(* Logix 5000 project; controller cal1632 1756-L62 rev 16.20; software revision 16.05; part 46 of 57 *)
(* tags used below, declared in another part *)
   FAULT : BOOL;
   HMI : BOOL;
   p01_recipe_active : recipe;
   p01r09_pb_global_reset : BOOL;
   p26_ao_dia_a : REAL;
   p26_ao_dia_b : REAL;
   p26_inactive_tension_sp : REAL;
   p26r03_upper_A_tension_on : BOOL;
   p26r03_upper_B_tension_on : BOOL;
   p26r10 : routine;
   p26r10_timer_fault : TIMER[4];
   p26r10_timer_warning : TIMER[4];
   p26r10_ula_selected_tension : REAL;
   p26r10_ulb_selected_tension : REAL;
   p26r10_unwind_a_brake_torque : REAL;
   p26r10_unwind_a_dia_ft : REAL;
   p26r10_unwind_b_brake_torque : REAL;
   p26r10_unwind_b_dia_ft : REAL;
   p27_ao_dia_a : REAL;
   p27_ao_dia_b : REAL;
   p27_dint_to_hmi : DINT[16];
   p27_lft_a_prs_input_max : REAL;
   p27_lft_a_prs_input_min : REAL;
   p27_lft_a_prs_output_max : REAL;
   p27_lft_a_prs_output_min : REAL;
   p27_lft_b_prs_input_max : REAL;
   p27_lft_b_prs_input_min : REAL;
   p27_lft_b_prs_output_max : REAL;
   p27_lft_b_prs_output_min : REAL;
   p27_lla_prs_input_max : REAL;
   p27_lla_prs_input_min : REAL;
   p27_lla_prs_output_max : REAL;
   p27_lla_prs_output_min : REAL;
   p27_lla_prs_scp : SYS_SCP;
   p27_llb_prs_input_max : REAL;
   p27_llb_prs_input_min : REAL;
   p27_llb_prs_output_max : REAL;
   p27_llb_prs_output_min : REAL;
   p27_llb_prs_scp : SYS_SCP;
   p27r01 : routine;
   p27r02 : routine;
   p27r02_fault_exists : BOOL;
   p27r02_timer_fault : TIMER[4];
   p27r02_timer_warning : TIMER[4];
   p27r02_unack_fault : BOOL;
   p27r02_unack_warning : BOOL;
   p27r02_warning_exists : BOOL;
   p27r03 : routine;
   p27r03_a_radius : REAL;
   p27r03_ai_dia_a_sensor : REAL;
   p27r03_ai_dia_b_sensor : REAL;
   p27r03_b_radius : REAL;
   p27r03_lower_A_tension_on : BOOL;
   p27r03_lower_B_tension_on : BOOL;
   p27r03_ltf_a_diameter_scp : SYS_SCP;
   p27r03_ltf_b_diameter_scp : SYS_SCP;
   p27r03_timer_fault : TIMER[4];
   p27r03_timer_warning : TIMER[4];
   p27r03_winder_a_distance : REAL;
   p27r03_winder_b_distance : REAL;
   p27r04 : routine;
   p27r04_timer_fault : TIMER[4];
   p27r04_timer_warning : TIMER[4];
   p27r05 : routine;
   p27r05_timer_fault : TIMER[4];
   p27r05_timer_warning : TIMER[4];
   p27r06 : routine;
   p27r07 : routine;
   p27r08 : routine;
   p27r09 : routine;
   p27r10 : routine;
   p27r10_lla_selected_tension : REAL;
   p27r10_llb_selected_tension : REAL;
   p27r11 : routine;
(* P26_Upper_Poly_Letoff, continued *)

ROUTINE R10_Tension_A   (* ladder *)
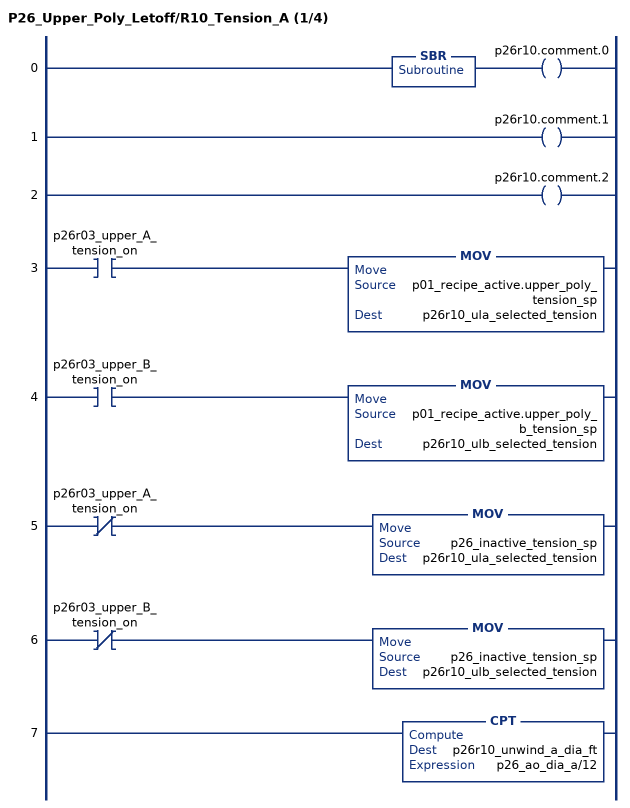
   0: SBR()OTE(p26r10.comment.0);
   1: OTE(p26r10.comment.1);
   2: OTE(p26r10.comment.2);
   3: XIC(p26r03_upper_A_tension_on)MOV(p01_recipe_active.upper_poly_tension_sp,p26r10_ula_selected_tension);
   4: XIC(p26r03_upper_B_tension_on)MOV(p01_recipe_active.upper_poly_b_tension_sp,p26r10_ulb_selected_tension);
   5: XIO(p26r03_upper_A_tension_on)MOV(p26_inactive_tension_sp,p26r10_ula_selected_tension);
   6: XIO(p26r03_upper_B_tension_on)MOV(p26_inactive_tension_sp,p26r10_ulb_selected_tension);
   7: CPT(p26r10_unwind_a_dia_ft,p26_ao_dia_a/12);
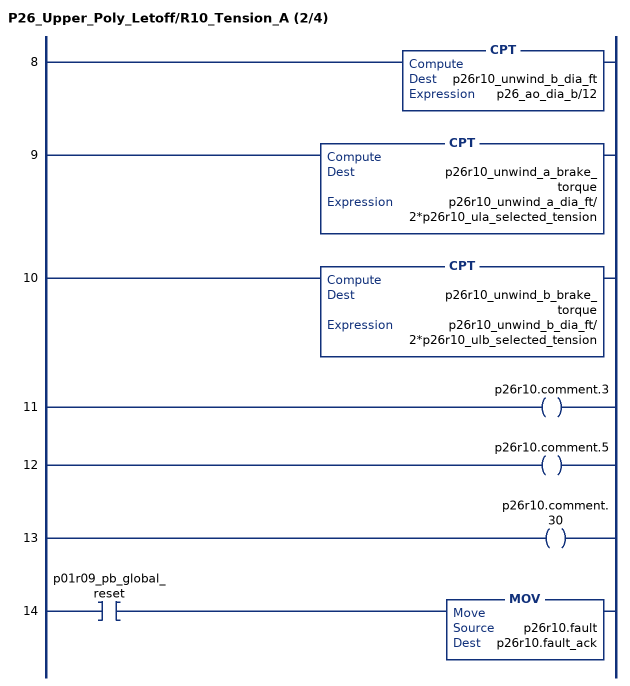
   8: CPT(p26r10_unwind_b_dia_ft,p26_ao_dia_b/12);
   9: CPT(p26r10_unwind_a_brake_torque,p26r10_unwind_a_dia_ft/2*p26r10_ula_selected_tension);
   10: CPT(p26r10_unwind_b_brake_torque,p26r10_unwind_b_dia_ft/2*p26r10_ulb_selected_tension);
   11: OTE(p26r10.comment.3);
   12: OTE(p26r10.comment.5);
   13: OTE(p26r10.comment.30);
   14: XIC(p01r09_pb_global_reset)MOV(p26r10.fault,p26r10.fault_ack);
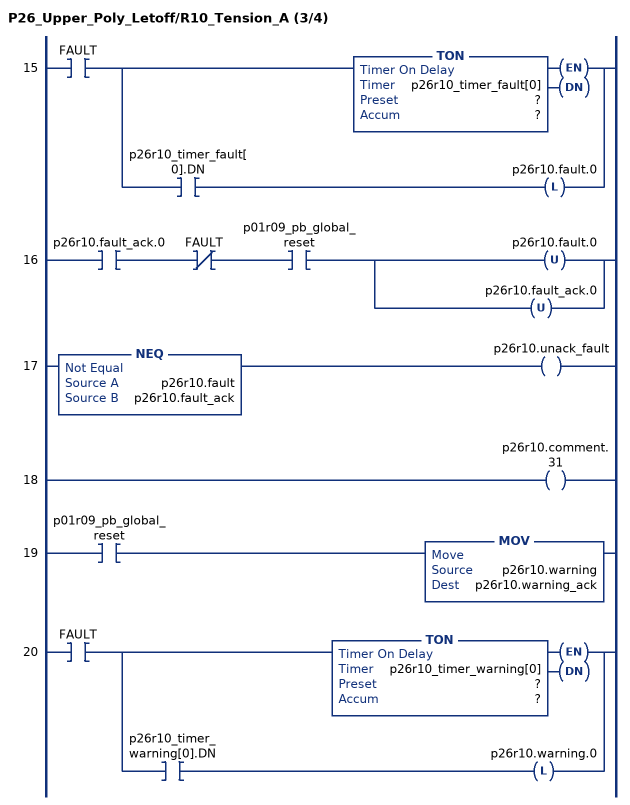
   15: XIC(FAULT)[TON(p26r10_timer_fault[0],?,?) ,XIC(p26r10_timer_fault[0].DN) OTL(p26r10.fault.0) ];
   16: XIC(p26r10.fault_ack.0)XIO(FAULT)XIC(p01r09_pb_global_reset)[OTU(p26r10.fault.0) ,OTU(p26r10.fault_ack.0) ];
   17: NEQ(p26r10.fault,p26r10.fault_ack)OTE(p26r10.unack_fault);
   18: OTE(p26r10.comment.31);
   19: XIC(p01r09_pb_global_reset)MOV(p26r10.warning,p26r10.warning_ack);
   20: XIC(FAULT)[TON(p26r10_timer_warning[0],?,?) ,XIC(p26r10_timer_warning[0].DN) OTL(p26r10.warning.0) ];
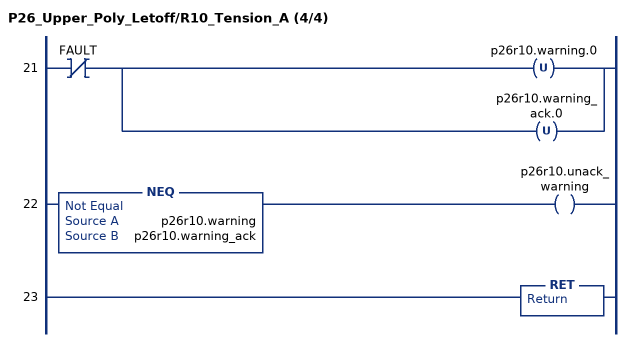
   21: XIO(FAULT)[OTU(p26r10.warning.0) ,OTU(p26r10.warning_ack.0) ];
   22: NEQ(p26r10.warning,p26r10.warning_ack)OTE(p26r10.unack_warning);
   23: RET();
END_ROUTINE
END_PROGRAM

PROGRAM P27_Lower_Poly_Letoff   (* main routine R01_Main *)

ROUTINE R01_Main   (* ladder *)
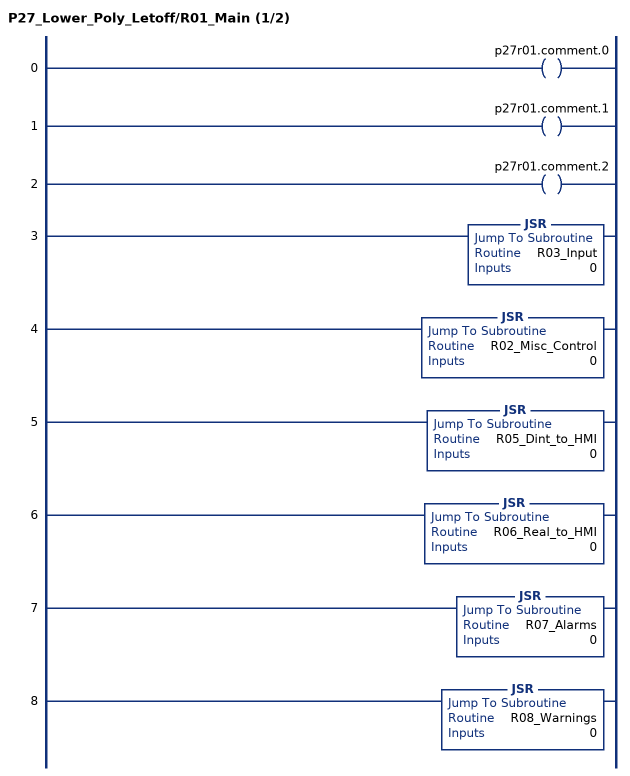
   0: OTE(p27r01.comment.0);
   1: OTE(p27r01.comment.1);
   2: OTE(p27r01.comment.2);
   3: JSR(R03_Input,0);
   4: JSR(R02_Misc_Control,0);
   5: JSR(R05_Dint_to_HMI,0);
   6: JSR(R06_Real_to_HMI,0);
   7: JSR(R07_Alarms,0);
   8: JSR(R08_Warnings,0);
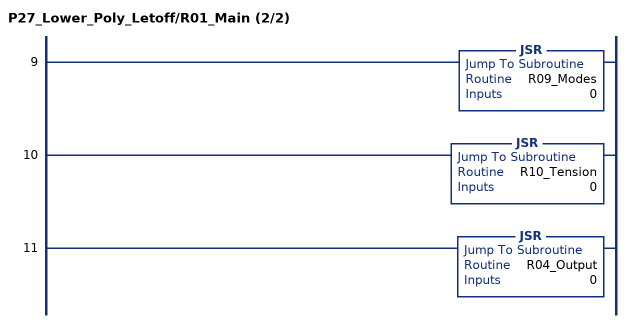
   9: JSR(R09_Modes,0);
   10: JSR(R10_Tension,0);
   11: JSR(R04_Output,0);
END_ROUTINE

ROUTINE R02_Misc_Control   (* ladder *)
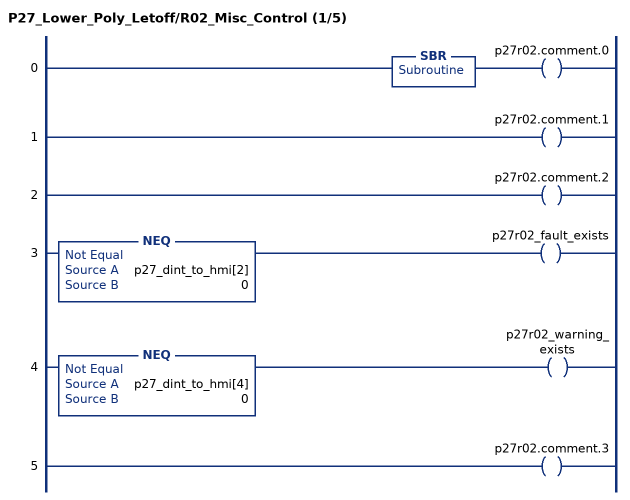
   0: SBR()OTE(p27r02.comment.0);
   1: OTE(p27r02.comment.1);
   2: OTE(p27r02.comment.2);
   3: NEQ(p27_dint_to_hmi[2],0)OTE(p27r02_fault_exists);
   4: NEQ(p27_dint_to_hmi[4],0)OTE(p27r02_warning_exists);
   5: OTE(p27r02.comment.3);
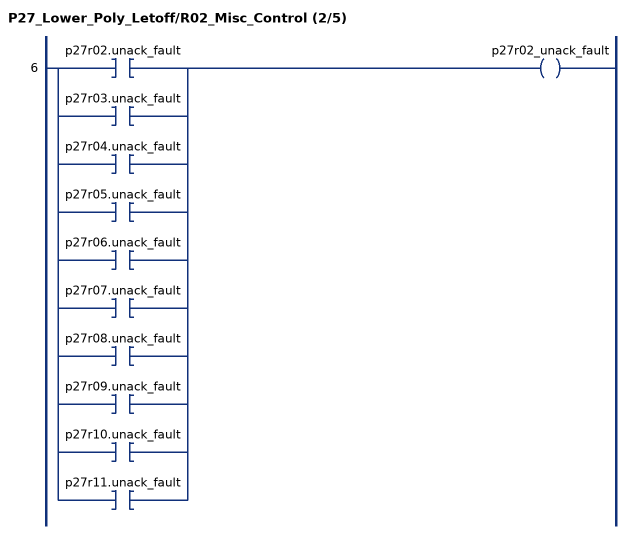
   6: [XIC(p27r02.unack_fault) ,XIC(p27r03.unack_fault) ,XIC(p27r04.unack_fault) ,XIC(p27r05.unack_fault) ,XIC(p27r06.unack_fault) ,XIC(p27r07.unack_fault) ,XIC(p27r08.unack_fault) ,XIC(p27r09.unack_fault) ,XIC(p27r10.unack_fault) ,XIC(p27r11.unack_fault) ]OTE(p27r02_unack_fault);
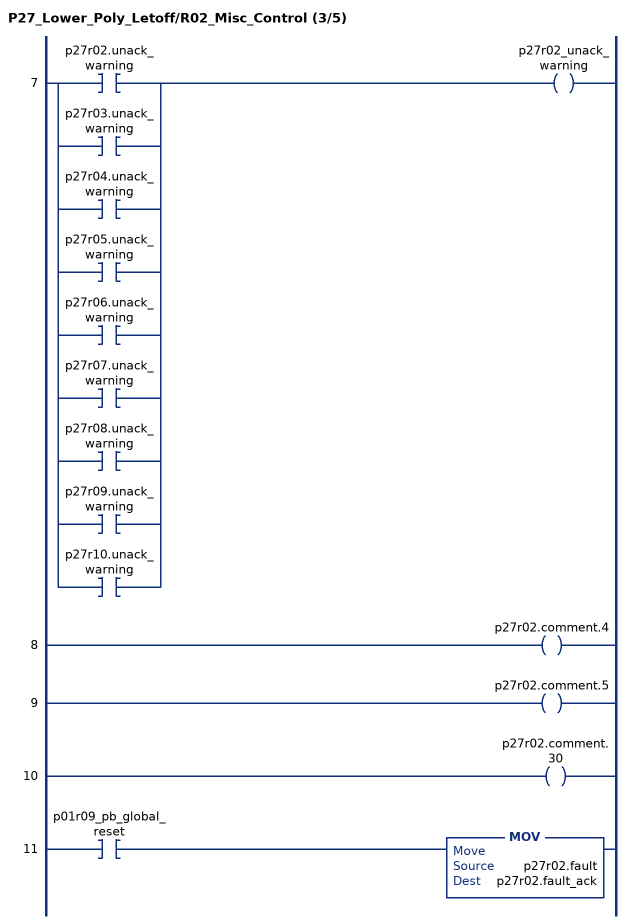
   7: [XIC(p27r02.unack_warning) ,XIC(p27r03.unack_warning) ,XIC(p27r04.unack_warning) ,XIC(p27r05.unack_warning) ,XIC(p27r06.unack_warning) ,XIC(p27r07.unack_warning) ,XIC(p27r08.unack_warning) ,XIC(p27r09.unack_warning) ,XIC(p27r10.unack_warning) ]OTE(p27r02_unack_warning);
   8: OTE(p27r02.comment.4);
   9: OTE(p27r02.comment.5);
   10: OTE(p27r02.comment.30);
   11: XIC(p01r09_pb_global_reset)MOV(p27r02.fault,p27r02.fault_ack);
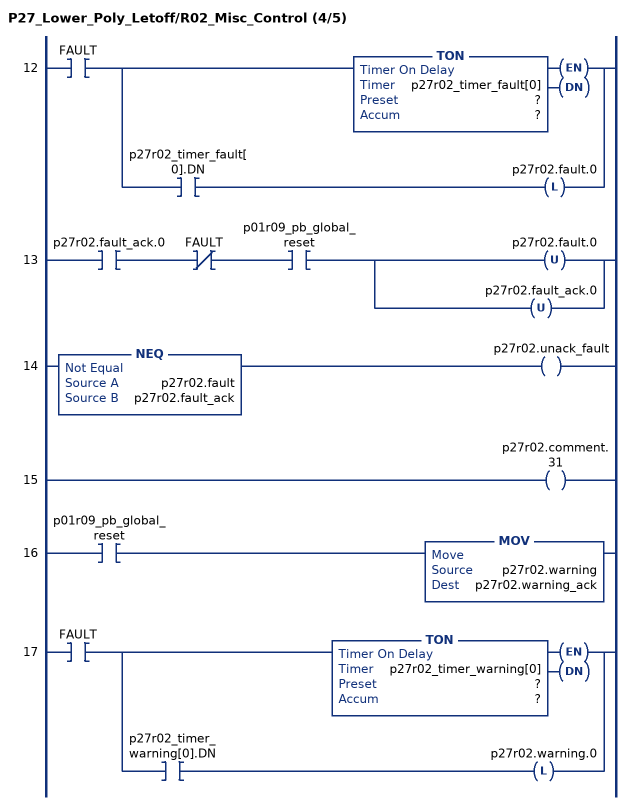
   12: XIC(FAULT)[TON(p27r02_timer_fault[0],?,?) ,XIC(p27r02_timer_fault[0].DN) OTL(p27r02.fault.0) ];
   13: XIC(p27r02.fault_ack.0)XIO(FAULT)XIC(p01r09_pb_global_reset)[OTU(p27r02.fault.0) ,OTU(p27r02.fault_ack.0) ];
   14: NEQ(p27r02.fault,p27r02.fault_ack)OTE(p27r02.unack_fault);
   15: OTE(p27r02.comment.31);
   16: XIC(p01r09_pb_global_reset)MOV(p27r02.warning,p27r02.warning_ack);
   17: XIC(FAULT)[TON(p27r02_timer_warning[0],?,?) ,XIC(p27r02_timer_warning[0].DN) OTL(p27r02.warning.0) ];
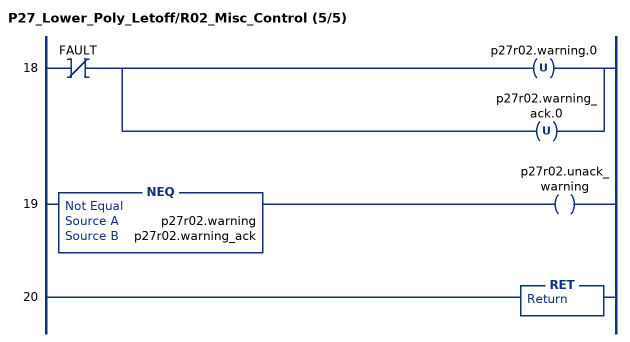
   18: XIO(FAULT)[OTU(p27r02.warning.0) ,OTU(p27r02.warning_ack.0) ];
   19: NEQ(p27r02.warning,p27r02.warning_ack)OTE(p27r02.unack_warning);
   20: RET();
END_ROUTINE

ROUTINE R03_Input   (* ladder *)
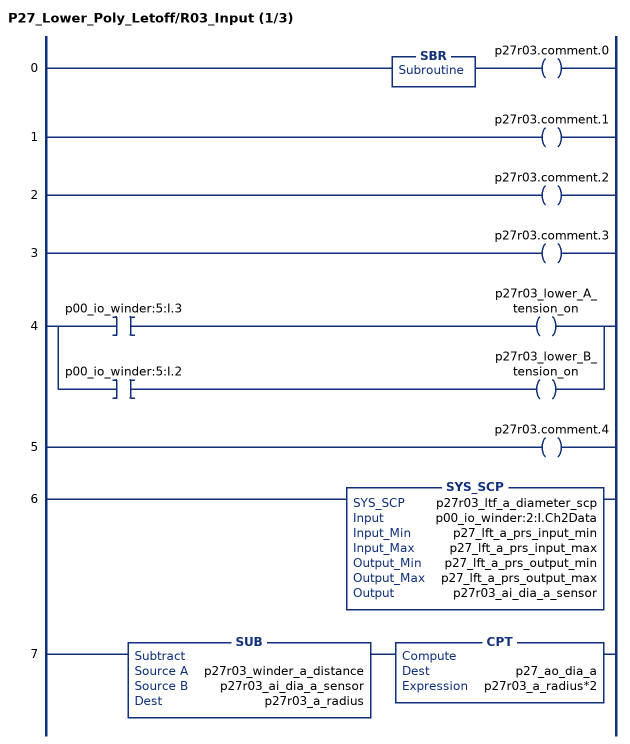
   0: SBR()OTE(p27r03.comment.0);
   1: OTE(p27r03.comment.1);
   2: OTE(p27r03.comment.2);
   3: OTE(p27r03.comment.3);
   4: [XIC(p00_io_winder:5:I.3) OTE(p27r03_lower_A_tension_on) ,XIC(p00_io_winder:5:I.2) OTE(p27r03_lower_B_tension_on) ];
   5: OTE(p27r03.comment.4);
   6: SYS_SCP(p27r03_ltf_a_diameter_scp,p00_io_winder:2:I.Ch2Data,p27_lft_a_prs_input_min,p27_lft_a_prs_input_max,p27_lft_a_prs_output_min,p27_lft_a_prs_output_max,p27r03_ai_dia_a_sensor);
   7: SUB(p27r03_winder_a_distance,p27r03_ai_dia_a_sensor,p27r03_a_radius)CPT(p27_ao_dia_a,p27r03_a_radius*2);
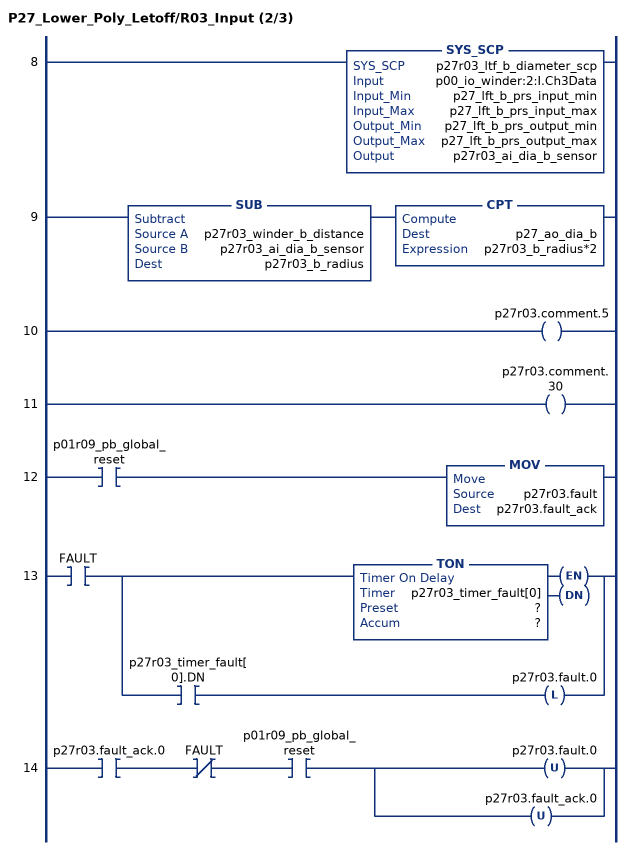
   8: SYS_SCP(p27r03_ltf_b_diameter_scp,p00_io_winder:2:I.Ch3Data,p27_lft_b_prs_input_min,p27_lft_b_prs_input_max,p27_lft_b_prs_output_min,p27_lft_b_prs_output_max,p27r03_ai_dia_b_sensor);
   9: SUB(p27r03_winder_b_distance,p27r03_ai_dia_b_sensor,p27r03_b_radius)CPT(p27_ao_dia_b,p27r03_b_radius*2);
   10: OTE(p27r03.comment.5);
   11: OTE(p27r03.comment.30);
   12: XIC(p01r09_pb_global_reset)MOV(p27r03.fault,p27r03.fault_ack);
   13: XIC(FAULT)[TON(p27r03_timer_fault[0],?,?) ,XIC(p27r03_timer_fault[0].DN) OTL(p27r03.fault.0) ];
   14: XIC(p27r03.fault_ack.0)XIO(FAULT)XIC(p01r09_pb_global_reset)[OTU(p27r03.fault.0) ,OTU(p27r03.fault_ack.0) ];
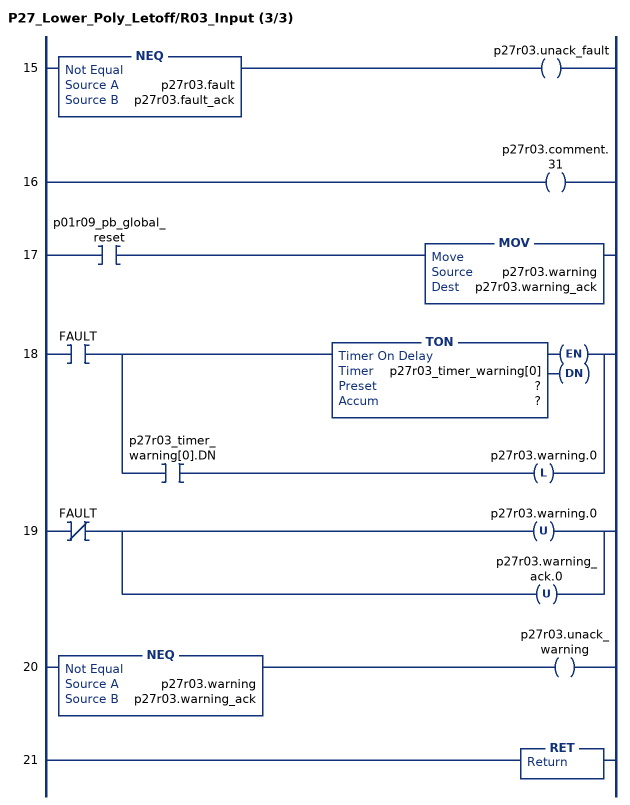
   15: NEQ(p27r03.fault,p27r03.fault_ack)OTE(p27r03.unack_fault);
   16: OTE(p27r03.comment.31);
   17: XIC(p01r09_pb_global_reset)MOV(p27r03.warning,p27r03.warning_ack);
   18: XIC(FAULT)[TON(p27r03_timer_warning[0],?,?) ,XIC(p27r03_timer_warning[0].DN) OTL(p27r03.warning.0) ];
   19: XIO(FAULT)[OTU(p27r03.warning.0) ,OTU(p27r03.warning_ack.0) ];
   20: NEQ(p27r03.warning,p27r03.warning_ack)OTE(p27r03.unack_warning);
   21: RET();
END_ROUTINE

ROUTINE R04_Output   (* ladder *)
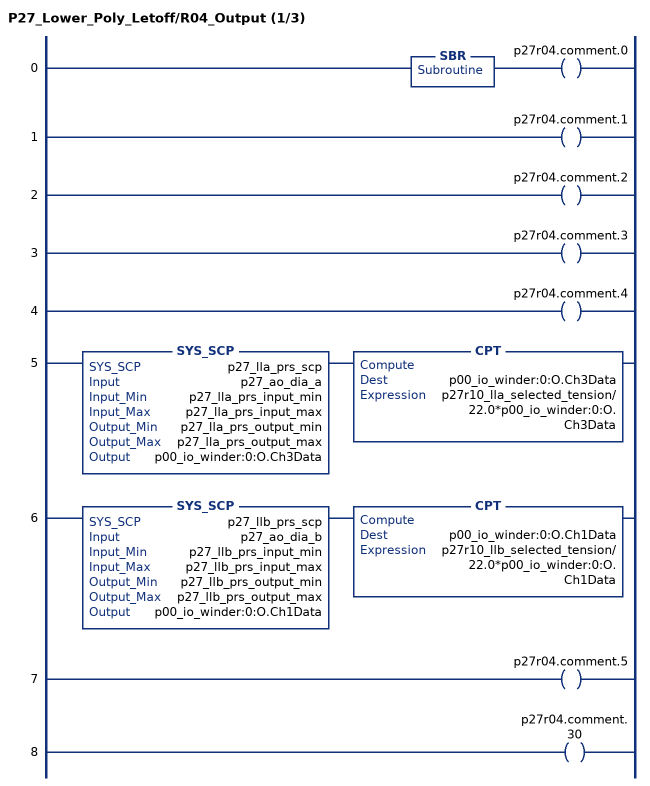
   0: SBR()OTE(p27r04.comment.0);
   1: OTE(p27r04.comment.1);
   2: OTE(p27r04.comment.2);
   3: OTE(p27r04.comment.3);
   4: OTE(p27r04.comment.4);
   5: SYS_SCP(p27_lla_prs_scp,p27_ao_dia_a,p27_lla_prs_input_min,p27_lla_prs_input_max,p27_lla_prs_output_min,p27_lla_prs_output_max,p00_io_winder:0:O.Ch3Data)CPT(p00_io_winder:0:O.Ch3Data,p27r10_lla_selected_tension/22.0*p00_io_winder:0:O.Ch3Data);
   6: SYS_SCP(p27_llb_prs_scp,p27_ao_dia_b,p27_llb_prs_input_min,p27_llb_prs_input_max,p27_llb_prs_output_min,p27_llb_prs_output_max,p00_io_winder:0:O.Ch1Data)CPT(p00_io_winder:0:O.Ch1Data,p27r10_llb_selected_tension/22.0*p00_io_winder:0:O.Ch1Data);
   7: OTE(p27r04.comment.5);
   8: OTE(p27r04.comment.30);
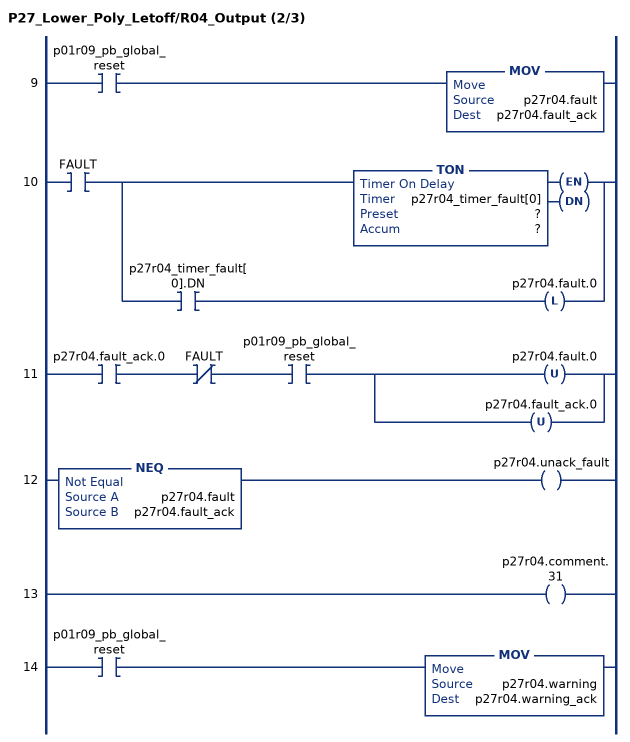
   9: XIC(p01r09_pb_global_reset)MOV(p27r04.fault,p27r04.fault_ack);
   10: XIC(FAULT)[TON(p27r04_timer_fault[0],?,?) ,XIC(p27r04_timer_fault[0].DN) OTL(p27r04.fault.0) ];
   11: XIC(p27r04.fault_ack.0)XIO(FAULT)XIC(p01r09_pb_global_reset)[OTU(p27r04.fault.0) ,OTU(p27r04.fault_ack.0) ];
   12: NEQ(p27r04.fault,p27r04.fault_ack)OTE(p27r04.unack_fault);
   13: OTE(p27r04.comment.31);
   14: XIC(p01r09_pb_global_reset)MOV(p27r04.warning,p27r04.warning_ack);
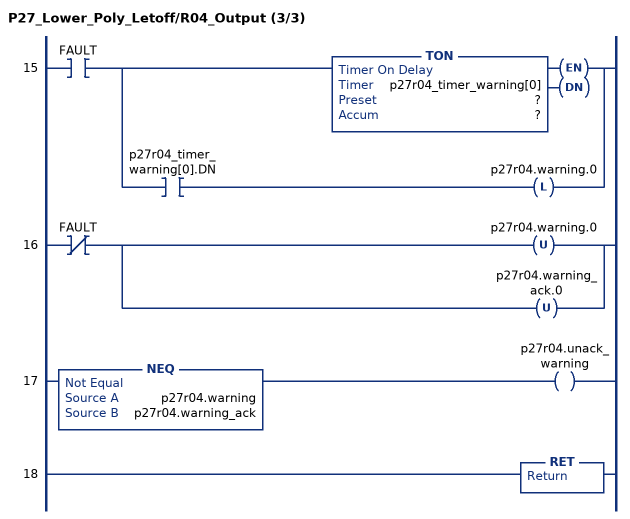
   15: XIC(FAULT)[TON(p27r04_timer_warning[0],?,?) ,XIC(p27r04_timer_warning[0].DN) OTL(p27r04.warning.0) ];
   16: XIO(FAULT)[OTU(p27r04.warning.0) ,OTU(p27r04.warning_ack.0) ];
   17: NEQ(p27r04.warning,p27r04.warning_ack)OTE(p27r04.unack_warning);
   18: RET();
END_ROUTINE

ROUTINE R05_Dint_to_HMI   (* ladder *)
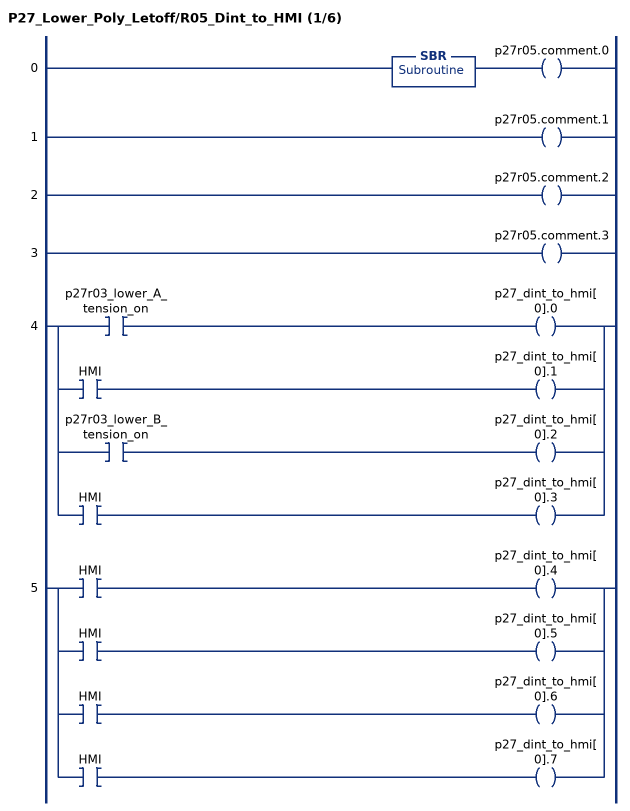
   0: SBR()OTE(p27r05.comment.0);
   1: OTE(p27r05.comment.1);
   2: OTE(p27r05.comment.2);
   3: OTE(p27r05.comment.3);
   4: [XIC(p27r03_lower_A_tension_on) OTE(p27_dint_to_hmi[0].0) ,XIC(HMI) OTE(p27_dint_to_hmi[0].1) ,XIC(p27r03_lower_B_tension_on) OTE(p27_dint_to_hmi[0].2) ,XIC(HMI) OTE(p27_dint_to_hmi[0].3) ];
   5: [XIC(HMI) OTE(p27_dint_to_hmi[0].4) ,XIC(HMI) OTE(p27_dint_to_hmi[0].5) ,XIC(HMI) OTE(p27_dint_to_hmi[0].6) ,XIC(HMI) OTE(p27_dint_to_hmi[0].7) ];
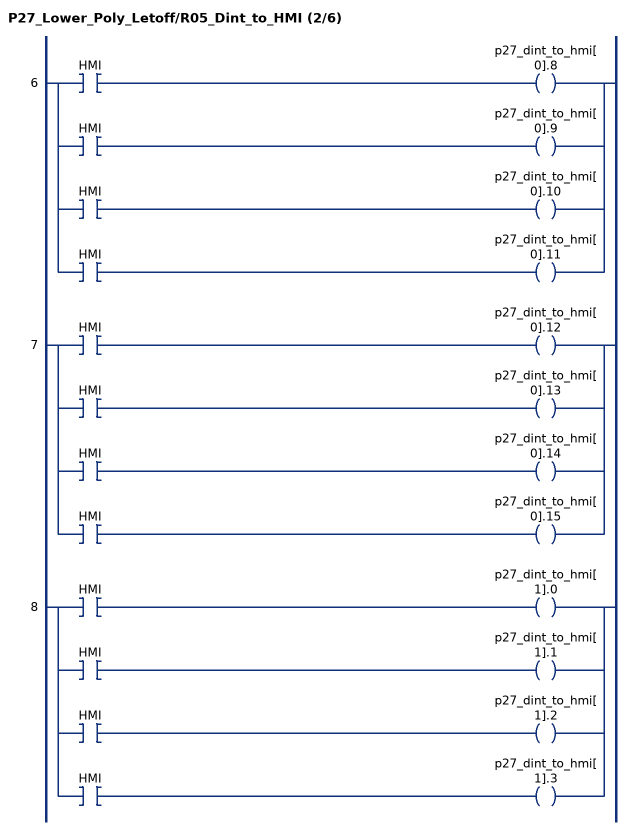
   6: [XIC(HMI) OTE(p27_dint_to_hmi[0].8) ,XIC(HMI) OTE(p27_dint_to_hmi[0].9) ,XIC(HMI) OTE(p27_dint_to_hmi[0].10) ,XIC(HMI) OTE(p27_dint_to_hmi[0].11) ];
   7: [XIC(HMI) OTE(p27_dint_to_hmi[0].12) ,XIC(HMI) OTE(p27_dint_to_hmi[0].13) ,XIC(HMI) OTE(p27_dint_to_hmi[0].14) ,XIC(HMI) OTE(p27_dint_to_hmi[0].15) ];
   8: [XIC(HMI) OTE(p27_dint_to_hmi[1].0) ,XIC(HMI) OTE(p27_dint_to_hmi[1].1) ,XIC(HMI) OTE(p27_dint_to_hmi[1].2) ,XIC(HMI) OTE(p27_dint_to_hmi[1].3) ];
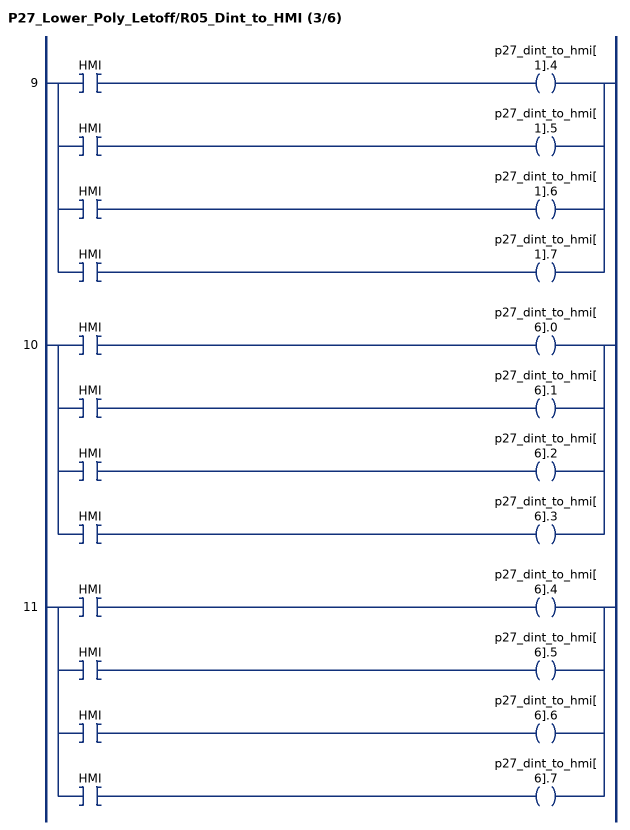
   9: [XIC(HMI) OTE(p27_dint_to_hmi[1].4) ,XIC(HMI) OTE(p27_dint_to_hmi[1].5) ,XIC(HMI) OTE(p27_dint_to_hmi[1].6) ,XIC(HMI) OTE(p27_dint_to_hmi[1].7) ];
   10: [XIC(HMI) OTE(p27_dint_to_hmi[6].0) ,XIC(HMI) OTE(p27_dint_to_hmi[6].1) ,XIC(HMI) OTE(p27_dint_to_hmi[6].2) ,XIC(HMI) OTE(p27_dint_to_hmi[6].3) ];
   11: [XIC(HMI) OTE(p27_dint_to_hmi[6].4) ,XIC(HMI) OTE(p27_dint_to_hmi[6].5) ,XIC(HMI) OTE(p27_dint_to_hmi[6].6) ,XIC(HMI) OTE(p27_dint_to_hmi[6].7) ];
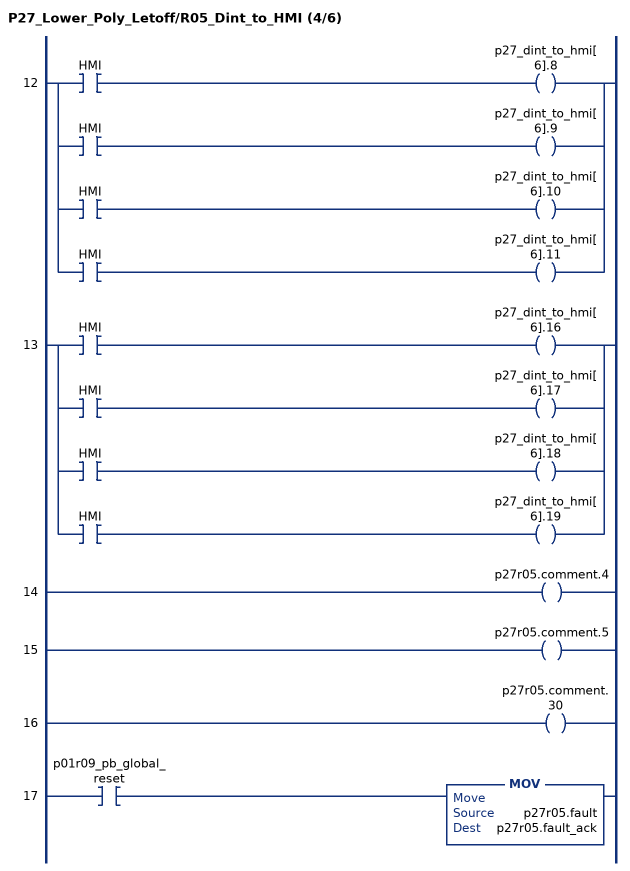
   12: [XIC(HMI) OTE(p27_dint_to_hmi[6].8) ,XIC(HMI) OTE(p27_dint_to_hmi[6].9) ,XIC(HMI) OTE(p27_dint_to_hmi[6].10) ,XIC(HMI) OTE(p27_dint_to_hmi[6].11) ];
   13: [XIC(HMI) OTE(p27_dint_to_hmi[6].16) ,XIC(HMI) OTE(p27_dint_to_hmi[6].17) ,XIC(HMI) OTE(p27_dint_to_hmi[6].18) ,XIC(HMI) OTE(p27_dint_to_hmi[6].19) ];
   14: OTE(p27r05.comment.4);
   15: OTE(p27r05.comment.5);
   16: OTE(p27r05.comment.30);
   17: XIC(p01r09_pb_global_reset)MOV(p27r05.fault,p27r05.fault_ack);
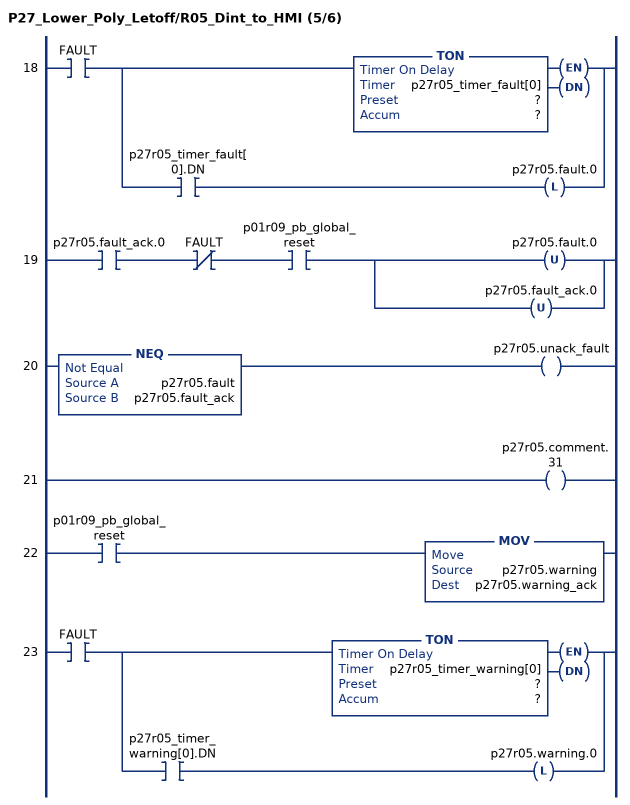
   18: XIC(FAULT)[TON(p27r05_timer_fault[0],?,?) ,XIC(p27r05_timer_fault[0].DN) OTL(p27r05.fault.0) ];
   19: XIC(p27r05.fault_ack.0)XIO(FAULT)XIC(p01r09_pb_global_reset)[OTU(p27r05.fault.0) ,OTU(p27r05.fault_ack.0) ];
   20: NEQ(p27r05.fault,p27r05.fault_ack)OTE(p27r05.unack_fault);
   21: OTE(p27r05.comment.31);
   22: XIC(p01r09_pb_global_reset)MOV(p27r05.warning,p27r05.warning_ack);
   23: XIC(FAULT)[TON(p27r05_timer_warning[0],?,?) ,XIC(p27r05_timer_warning[0].DN) OTL(p27r05.warning.0) ];
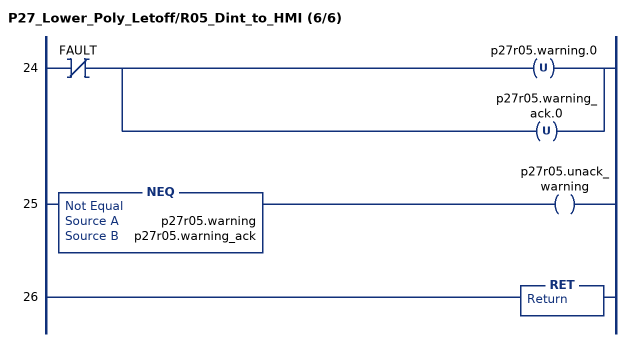
   24: XIO(FAULT)[OTU(p27r05.warning.0) ,OTU(p27r05.warning_ack.0) ];
   25: NEQ(p27r05.warning,p27r05.warning_ack)OTE(p27r05.unack_warning);
   26: RET();
END_ROUTINE
